(* CODESYS project DCCM PLC 1.project
   Author: jrfsc
   Version: 0.0.0.0
   Title: DCCM PLC 1

Project tree, tasks and I/O mapping:
  DCCM_PLC_1 : TM251MESC, Schneider Electric, order no. TM251MESC, version 5.1.9.35
      settings: OPCUA enable = False
    application Application
      libraries: SysTimeRtc, * (System); CAA Memory, 3.5.12.0 (CAA Technical Workgroup); IecRtsServices, 1.0.4.0 (Schneider Electric)
      task MAST (cyclic, interval 20 ms, priority 15, watchdog 100 ms x 1) calls INPUT_MAPPING, FILTER_ALARMS, FAN_2STAGES_FAULT_DETECTION, DEPROX_COUNT, FAN_2STAGES, PandemicCheck, DAMPER_CONTROL, SR_Main, OUTPUT_MAPPING
      global variables GVL
      program SR_Main [FBD]
      program INPUT_MAPPING [ST]
      program OUTPUT_MAPPING [ST]
      FBs/
        function block DUTY [ST]
        function block DUTY_CHANGE [ST]
        function block FB_9StatesMonitoring [ST]
        function block FB_DUTY_DUTY_STANDBY_PUMP_SPD [ST]
        function block FB_FLOATING_VALVE [ST]
        function block FB_HEATING_OR_COOLING [ST]
        function block FB_OMODE [ST]
        function block FB_PMODE [ST]
        function block FB_SETPOINT_MODE [ST]
        function block FB_WATCHDOG [ST]
        function block LINEAR [ST]
        function block SATSP_CALC [ST]
        function block SB_HEATING_COOLING [ST]
        function block TERMINAL_LOAD [ST]
        function block FB_0_10V_TO_2_10V_OUTPUT [ST]
        function block FB_2STAGES_DUTY [ST]
        function block FB_DUTYTRIGGER [ST]
        function block FB_FanProvingSwitchOverEnable [ST]
        function block FB_2STAGES_DUTY_1 [ST]
        function block SWITCH_CHECK [ST]
      Enumeration/
        data type ET_9STATE_MONITORING
        data type ET_OMODE
        data type ET_PMODE
      LIBRARY/
        function block FB_PULSE_GENERATOR [ST]
      Library/
        function block FB_SETPOINT_RAMPING [ST]
        function block FB_PCMS_WATCHDOG [ST]
      program SYSTEM_DATE_TIME [ST]
      program DAMPER_CONTROL [FBD]
      program FILTER_ALARMS [FBD]
      program DEPROX_COUNT [CFC]
      program FAN_2STAGES [FBD]: ACT_GetCurrentDateTime
      program FAN_2STAGES_FAULT_DETECTION [FBD]
      global variables PersistentVars
      program PandemicCheck [CFC]
    IO_Bus : IO bus - TM3, Schneider Electric, version 5.1.9.35
      Module_1 : TM3AQ4/G, Schneider Electric, order no. TM3AQ4/G, version 1.0.0.16
          settings: KPI Configuration.KPI Configuration = 16; KPI Configuration.KPI Configuration = 0; KPI Configuration.KPI Configuration = 16; KPI Configuration.KPI Configuration = 39
          output qPLANT_EXHAUST_DAMPER : INT  // QW0
          output qiModule_1_QW3 : INT  // QW3
          input  ibModule_1_IBStatusQW0 : BYTE  // IBStatusQW0
          input  ibModule_1_IBStatusQW1 : BYTE  // IBStatusQW1
          input  ibModule_1_IBStatusQW2 : BYTE  // IBStatusQW2
          input  ibModule_1_IBStatusQW3 : BYTE  // IBStatusQW3
          unmapped channels: QW1, QW2
      Module_2 : TM3AI8/G, Schneider Electric, order no. TM3AI8/G, version 1.0.0.27
          settings: KPI Configuration.KPI Configuration = 32; KPI Configuration.KPI Configuration = 32; KPI Configuration.KPI Configuration = 32; KPI Configuration.KPI Configuration = 32; KPI Configuration.KPI Configuration = 32; KPI Configuration.KPI Configuration = 32; KPI Configuration.KPI Configuration = 32; KPI Configuration.KPI Configuration = 32; KPI Configuration.KPI Configuration = 0; KPI Configuration.KPI Configuration = 0; KPI Configuration.KPI Configuration = 0; KPI Configuration.KPI Configuration = 0; KPI Configuration.KPI Configuration = 0; KPI Configuration.KPI Configuration = 0; KPI Configuration.KPI Configuration = 0; KPI Configuration.KPI Configuration = 0; KPI Configuration.KPI Configuration = 50; KPI Configuration.KPI Configuration = 0; KPI Configuration.KPI Configuration = 250; KPI Configuration.KPI Configuration = 0; KPI Configuration.KPI Configuration = 250; KPI Configuration.KPI Configuration = 0; KPI Configuration.KPI Configuration = 250; KPI Configuration.KPI Configuration = 0; KPI Configuration.KPI Configuration = 244; KPI Configuration.KPI Configuration = 1; KPI Configuration.KPI Configuration = 244; KPI Configuration.KPI Configuration = 1; KPI Configuration.KPI Configuration = 244; KPI Configuration.KPI Configuration = 1; KPI Configuration.KPI Configuration = 16; KPI Configuration.KPI Configuration = 39; KPI Configuration.KPI Configuration = 100
          input  iEXHAUST_AIR_VELOCITY : INT  // IW0
          input  iPREFILTER1_DP : INT  // IW1
          input  iPREFILTER2_DP : INT  // IW2
          input  iPREFILTER3_DP : INT  // IW3
          input  iHEPA1_DP : INT  // IW4
          input  iHEPA2_DP : INT  // IW5
          input  iHEPA3_DP : INT  // IW6
          input  iPLANT_EXHAUST_DAMPER_STS : INT  // IW7
          input  ibModule_2_IBStatusIW0 : BYTE  // IBStatusIW0
          input  ibModule_2_IBStatusIW1 : BYTE  // IBStatusIW1
          input  ibModule_2_IBStatusIW2 : BYTE  // IBStatusIW2
          input  ibModule_2_IBStatusIW3 : BYTE  // IBStatusIW3
          input  ibModule_2_IBStatusIW4 : BYTE  // IBStatusIW4
          input  ibModule_2_IBStatusIW5 : BYTE  // IBStatusIW5
          input  ibModule_2_IBStatusIW6 : BYTE  // IBStatusIW6
          input  ibModule_2_IBStatusIW7 : BYTE  // IBStatusIW7
      Module_3 : TM3DM24R/G, Schneider Electric, order no. TM3DM24R/G, version 1.0.2.0
          input  iPRESSURE_SWITCH1 : BOOL  // IW0.I0
          input  iPRESSURE_SWITCH2 : BOOL  // IW0.I1
          input  iFAN1_MANUAL_SW : BOOL  // IW0.I2
          input  iFAN1_AUTO_SW : BOOL  // IW0.I3
          input  iFAN2_MANUAL_SW : BOOL  // IW0.I4
          input  iFAN2_AUTO_SW : BOOL  // IW0.I5
          input  iFAN1_READY : BOOL  // IW0.I6
          input  iFAN1_RUN : BOOL  // IW0.I7
          input  iFAN1_FAULT : BOOL  // IW0.I8
          input  iFAN2_READY : BOOL  // IW0.I9
          input  iFAN2_RUN : BOOL  // IW0.I10
          input  iFAN2_FAULT : BOOL  // IW0.I11
          input  iFIRE_DAMPER_STS : BOOL  // IW0.I12
          input  iDISCHARGE_DAMPER1_STS : BOOL  // IW0.I13
          input  iDISCHARGE_DAMPER2_STS : BOOL  // IW0.I14
          input  iRETURN_DAMPER1_STS : BOOL  // IW0.I15
          output qFAN1_SS : BOOL  // QB0.Q0
          output qFAN2_SS : BOOL  // QB0.Q1
          output qFAN1_DISCHARGE_DAMPER : BOOL  // QB0.Q2
          output qFAN2_DISCHARGE_DAMPER : BOOL  // QB0.Q3
          output qPLANT_RETURN_DAMPER : BOOL  // QB0.Q4
          unmapped channels: IW0, QB0
      Module_4 : TM3AM6/G, Schneider Electric, order no. TM3AM6/G, version 1.0.0.23
          settings: KPI Configuration.KPI Configuration = 32; KPI Configuration.KPI Configuration = 32; KPI Configuration.KPI Configuration = 0; KPI Configuration.KPI Configuration = 0; KPI Configuration.KPI Configuration = 16; KPI Configuration.KPI Configuration = 39; KPI Configuration.KPI Configuration = 16; KPI Configuration.KPI Configuration = 39; KPI Configuration.KPI Configuration = 16; KPI Configuration.KPI Configuration = 16; KPI Configuration.KPI Configuration = 0; KPI Configuration.KPI Configuration = 0; KPI Configuration.KPI Configuration = 16; KPI Configuration.KPI Configuration = 39; KPI Configuration.KPI Configuration = 16; KPI Configuration.KPI Configuration = 39
          input  iFAN1_SPDFB : INT  // IW0
          input  iFAN2_SPDFB : INT  // IW1
          input  iiModule_4_IW2 : INT  // IW2
          input  iiModule_4_IW3 : INT  // IW3
          output qFAN1_SPD : INT  // QW0
          output qFAN2_SPD : INT  // QW1
          input  ibModule_4_IBStatusIW0 : BYTE  // IBStatusIW0
          input  ibModule_4_IBStatusIW1 : BYTE  // IBStatusIW1
          input  ibModule_4_IBStatusIW2 : BYTE  // IBStatusIW2
          input  ibModule_4_IBStatusIW3 : BYTE  // IBStatusIW3
          input  ibModule_4_IBStatusQW0 : BYTE  // IBStatusQW0
          input  ibModule_4_IBStatusQW1 : BYTE  // IBStatusQW1
    COM_Bus : COM bus, Schneider Electric, version 5.1.9.35
    Ethernet_1 : Ethernet Network, Schneider Electric, version 5.1.9.35
        settings: WebServer = TRUE; FTP Server = FALSE; SoMachine Protocol = TRUE; Modbus Server = TRUE; NetManage Protocol = TRUE; SNMP protocol = FALSE; WebVisu protocol = FALSE; Secured Web Server = TRUE
    Serial_Line_1 : Serial line, Schneider Electric, version 5.1.9.35
      Machine_Expert_Network_Manager : Machine Expert-Network Manager, Schneider Electric, version 4.0.0.4
    CAN_1 : CANopen bus, Schneider Electric, version 5.1.9.35
  FdtConnections : FDT Connections, Schneider Electric, version 1.0.0.2
*)

// DCCM_PLC_1/Application/Enumeration/ET_9STATE_MONITORING
{attribute 'qualified_only' := ''}
{attribute 'strict' := ''}
TYPE ET_9STATE_MONITORING :
(
	STOPPED := 0,
	RUNNING := 1,
	STARTING := 2,
	STOPPING := 3,
	START_FAIL := 4,
	STOP_FAIL := 5,
	UNEXPECTED_START := 6,
	UNEXPECTED_STOP := 7,
	FIRE_STOP := 8,
	UNKNOWN := 9
);
END_TYPE

// DCCM_PLC_1/Application/Enumeration/ET_OMODE
{attribute 'qualified_only' := ''}
{attribute 'strict' := ''}
TYPE ET_OMODE :
(
	UNOCC := 0,
	OPTSTART := 1,
	SCH := 2,
	AHRS := 3,
	MOTDETECT := 4,
	SETBACK := 7
);
END_TYPE

// DCCM_PLC_1/Application/Enumeration/ET_PMODE
{attribute 'qualified_only' := ''}
{attribute 'strict' := ''}
TYPE ET_PMODE :
(
	OFF_NORMAL := 0,
	OFF_PCMS := 1,
	OFF_Fire := 2,
	OFF_DMPRLOCK := 3,
	OFF_RESET := 4,
	Startup := 5,
	Purge := 6,
	RUN_NORMAL := 7
);
END_TYPE

// DCCM_PLC_1/Application/GVL
{attribute 'qualified_only'}
VAR_GLOBAL
	FAN1_SPEED AT %MD500: REAL;
	FAN2_SPEED AT %MD501: REAL;
	COMMS_ERROR_ROOM AT %MX6.1: BOOL;
	FAN2_FB AT %MD534: REAL;
	FAN1_FB AT %MD533: REAL;
	FAN1_SWITCH_TOTAL AT %MW9006: INT;
	FAN2_SWITCH_TOTAL AT %MW9007: INT;
	fan2SS_del: BOOL;
	fan1SS_del: bool;
	VEL_PRESS_LITRES AT %MD536: REAL;
	FAN2_FAULT_RESET AT %MX5.7: BOOL;
	FAN1_FAULT_RESET AT %MX5.6: BOOL;
END_VAR
VAR_GLOBAL RETAIN PERSISTENT
	EXHAUST_VEL_PRESS_SP AT %MD502: REAL := 3;
END_VAR
VAR_GLOBAL
	PREFILTER1_DP AT %MD503: REAL;
	PREFILTER2_DP AT %MD504: REAL;
	PREFILTER3_DP AT %MD505: REAL;
	HEPA1_DP AT %MD506: REAL;
	HEPA2_DP AT %MD507: REAL;
	HEPA3_DP AT %MD508: REAL;
	PRESSURE_SWITCH1 AT %MX0.0: BOOL;
	PRESSURE_SWITCH2 AT %MX0.1: BOOL;
	FAN1_MANUAL_SW AT %MX0.2: BOOL;
	FAN1_AUTO_SW AT %MX0.3: BOOL;
	FAN2_MANUAL_SW AT %MX0.4: BOOL;
	FAN2_AUTO_SW AT %MX0.5: BOOL;
	FAN1_READY AT %MX0.6: BOOL;
	FAN1_RUN AT %MX0.7: BOOL;
	FAN1_FAULT AT %MX1.0: BOOL;
	FAN2_READY AT %MX1.1: BOOL;
	FAN2_RUN AT %MX1.2: BOOL;
	FAN2_FAULT AT %MX1.3: BOOL;
	FIRE AT %MX1.4: BOOL;
	DISCHARGE_DAMPER1_STS AT %MX1.5: BOOL;
	DISCHARGE_DAMPER2_STS AT %MX1.6: BOOL;
	FAN1_SS AT %MX1.7: BOOL;
	FAN2_SS AT %MX2.0: BOOL;
	FAN1_DISCHARGE_DAMPER AT %MX2.1: BOOL;
	FAN2_DISCHARGE_DAMPER AT %MX2.2: BOOL;
	SYS_HOUR: UINT;
	SYS_DAY: UINT;
	SYS_MINUTE: UINT;
END_VAR
VAR_GLOBAL RETAIN PERSISTENT
	STANDBY_FAN_NO AT %MW9002: INT := 2;
	STANDBY_FAN_NO_MANUAL AT %MW9003: INT := 1;
	STANDBY_FAN_NO_MODE AT %MX2.5: BOOL := 1;
	FAN1_SS_MANUAL AT %MX2.6: BOOL;
	FAN1_SS_MODE AT %MX2.7: BOOL;
	FAN2_SS_MANUAL AT %MX3.0: BOOL;
	FAN2_SS_MODE AT %MX3.1: BOOL;
END_VAR
VAR_GLOBAL
	EXHAUST_VEL_PRESS AT %MD509: REAL;
END_VAR
VAR_GLOBAL RETAIN PERSISTENT
	FAN1_SPEED_MANUAL AT %MD510: REAL;
	FAN1_SPEED_MODE AT %MX3.2: BOOL;
	FAN2_SPEED_MANUAL AT %MD511: REAL;
	FAN2_SPEED_MODE AT %MX4.5: BOOL;
END_VAR
VAR_GLOBAL
	ISO_MD1 AT %MD527: REAL;
END_VAR
VAR_GLOBAL RETAIN PERSISTENT
	EF_VEL_PRESS_SP1 AT %MD512: REAL := 2;
	FAN1_DISCHARGE_DAMPER_MAN AT %MX3.3: BOOL;
	FAN1_DISCHARGE_DAMPER_MD AT %MX3.4: BOOL;
	FAN2_DISCHARGE_DAMPER_MAN AT %MX3.5: BOOL;
	FAN2_DISCHARGE_DAMPER_MD AT %MX3.6: BOOL;
END_VAR
VAR_GLOBAL
	FAN1_ST_MONITORING AT %MW9001: UINT;
	FAN2_ST_MONITORING AT %MW9004: UINT;
END_VAR
VAR_GLOBAL RETAIN PERSISTENT
	PREFILTER1_ALMSP AT %MD513: REAL;
	PREFILTER2_ALMSP AT %MD514: REAL;
	PREFILTER3_ALMSP AT %MD515: REAL;
	HEPA1_ALMSP AT %MD516: REAL;
	HEPA2_ALMSP AT %MD517: REAL;
	HEPA3_ALMSP AT %MD518: REAL;
END_VAR
VAR_GLOBAL
	PREFILTER1_ALM AT %MX3.7: BOOL;
	PREFILTER2_ALM AT %MX4.0: BOOL;
	PREFILTER3_ALM AT %MX4.1: BOOL;
	HEPA1_ALM AT %MX4.2: BOOL;
	HEPA2_ALM AT %MX4.3: BOOL;
	HEPA3_ALM AT %MX4.4: BOOL;
	ISO_MD2 AT %MD524: REAL;
	ISO_MD3 AT %MD525: REAL;
	ISO_MD4 AT %MD526: REAL;
	ISO_MD1_DW: REAL;
	ISO_MD2_DW: REAL;
	ISO_MD3_DW: REAL;
	ISO_MD4_DW: REAL;
END_VAR
VAR_GLOBAL RETAIN PERSISTENT
	PLANT_EXHAUST_DAMPER AT %MD523: REAL;
	PLANT_RETURN_DAMPER AT %MX5.2: BOOL;
	PLANT_RETURN_DAMPER_STS AT %MX5.1: BOOL;
END_VAR
VAR_GLOBAL
	PLANT_EXHAUST_DAMPER_STS AT %MD522: REAL;
END_VAR
VAR_GLOBAL RETAIN PERSISTENT
	PLANT_RETURN_DAMPER_MAN AT %MX5.0: BOOL;
	PLANT_RETURN_DAMPER_MD AT %MX5.5: BOOL;
	PLANT_RETURN_DAMPER_SS AT %MX5.4: BOOL;
	PLANT_EXHAUST_DAMPER_MD AT %MX5.3: BOOL;
	PLANT_EXHAUST_DAMPER_MAN AT %MD520: REAL;
	PLANT_EXHAUST_DAMPER_PAN AT %MD535: REAL;
	PLANT_EXHAUST_DAMPER_SP AT %MD521: REAL := 100;
	EF_VEL_PRESS_SP2 AT %MD528: REAL := 2;
	EF_VEL_PRESS_SP3 AT %MD529: REAL := 2;
	EF_VEL_PRESS_SP4 AT %MD530: REAL := 0;
	FAN_PID_P AT %MD532: REAL;
	FAN_PID_I AT %MD531: REAL;
	EXHAUST_VEL_PRESS_PAN_SP AT %MD550: REAL := 16;
	EXHAUST_VEL_PRESS_PAN_SP1 AT %MD551: REAL := 14;
	EXHAUST_VEL_PRESS_PAN_SP2 AT %MD552: REAL := 10;
	EXHAUST_VEL_PRESS_PAN_SP3 AT %MD553: REAL := 8;
	EXHAUST_VEL_PRESS_PAN_SP4 AT %MD554: REAL := 0;
END_VAR
VAR_GLOBAL
	OPEN_DAMPER1: BOOL;
	OPEN_DAMPER2: BOOL;
	FAN1_ST: BOOL;
	FAN2_ST: BOOL;
	PANDEMIC AT %MW9005: INT;
	COMMS_ERROR: BOOL;
	newVarGlobal: BOOL;
	COMMS_ERROR_AHU AT %MX6.0: BOOL;
END_VAR

// DCCM_PLC_1/Application/PersistentVars
{attribute 'qualified_only'}
VAR_GLOBAL PERSISTENT RETAIN
	// Generated instance path of persistent variable
	GVL.EXHAUST_VEL_PRESS_SP: REAL;
	// Generated instance path of persistent variable
	GVL.STANDBY_FAN_NO: INT := INT#2;
	// Generated instance path of persistent variable
	GVL.STANDBY_FAN_NO_MANUAL: INT := INT#1;
	// Generated instance path of persistent variable
	GVL.STANDBY_FAN_NO_MODE: BOOL := TRUE;
	// Generated instance path of persistent variable
	GVL.FAN1_SS_MANUAL: BOOL;
	// Generated instance path of persistent variable
	GVL.FAN1_SS_MODE: BOOL;
	// Generated instance path of persistent variable
	GVL.FAN2_SS_MANUAL: BOOL;
	// Generated instance path of persistent variable
	GVL.FAN2_SS_MODE: BOOL;
	// Generated instance path of persistent variable
	GVL.FAN1_SPEED_MANUAL: REAL;
	// Generated instance path of persistent variable
	GVL.FAN1_SPEED_MODE: BOOL;
	// Generated instance path of persistent variable
	GVL.FAN2_SPEED_MANUAL: REAL;
	// Generated instance path of persistent variable
	GVL.FAN2_SPEED_MODE: BOOL;
	// Generated instance path of persistent variable
	GVL.EF_VEL_PRESS_SP1: REAL;
	// Generated instance path of persistent variable
	GVL.FAN1_DISCHARGE_DAMPER_MAN: BOOL;
	// Generated instance path of persistent variable
	GVL.FAN1_DISCHARGE_DAMPER_MD: BOOL;
	// Generated instance path of persistent variable
	GVL.FAN2_DISCHARGE_DAMPER_MAN: BOOL;
	// Generated instance path of persistent variable
	GVL.FAN2_DISCHARGE_DAMPER_MD: BOOL;
	// Generated instance path of persistent variable
	GVL.PREFILTER1_ALMSP: REAL;
	// Generated instance path of persistent variable
	GVL.PREFILTER2_ALMSP: REAL;
	// Generated instance path of persistent variable
	GVL.PREFILTER3_ALMSP: REAL;
	// Generated instance path of persistent variable
	GVL.HEPA1_ALMSP: REAL;
	// Generated instance path of persistent variable
	GVL.HEPA2_ALMSP: REAL;
	// Generated instance path of persistent variable
	GVL.HEPA3_ALMSP: REAL;
	// Generated instance path of persistent variable
	GVL.PLANT_EXHAUST_DAMPER: REAL;
	// Generated instance path of persistent variable
	GVL.PLANT_RETURN_DAMPER: BOOL;
	// Generated instance path of persistent variable
	GVL.PLANT_RETURN_DAMPER_STS: BOOL;
	// Generated instance path of persistent variable
	GVL.PLANT_RETURN_DAMPER_MAN: BOOL;
	// Generated instance path of persistent variable
	GVL.PLANT_RETURN_DAMPER_MD: BOOL;
	// Generated instance path of persistent variable
	GVL.PLANT_RETURN_DAMPER_SS: BOOL;
	// Generated instance path of persistent variable
	GVL.PLANT_EXHAUST_DAMPER_MD: BOOL;
	// Generated instance path of persistent variable
	GVL.PLANT_EXHAUST_DAMPER_MAN: REAL;
	// Generated instance path of persistent variable
	GVL.PLANT_EXHAUST_DAMPER_PAN: REAL;
	// Generated instance path of persistent variable
	GVL.PLANT_EXHAUST_DAMPER_SP: REAL := 100.0;
	// Generated instance path of persistent variable
	GVL.EF_VEL_PRESS_SP2: REAL;
	// Generated instance path of persistent variable
	GVL.EF_VEL_PRESS_SP3: REAL;
	// Generated instance path of persistent variable
	GVL.EF_VEL_PRESS_SP4: REAL;
	// Generated instance path of persistent variable
	GVL.FAN_PID_P: REAL;
	// Generated instance path of persistent variable
	GVL.FAN_PID_I: REAL;
END_VAR

// DCCM_PLC_1/Application/INPUT_MAPPING
PROGRAM INPUT_MAPPING
VAR

	voltage_converter: FB_0_10V_TO_2_10V_OUTPUT;
END_VAR

//MAPPINGHARDWARE INPUTS TO MEMORY WORDS

GVL.EXHAUST_VEL_PRESS := TO_REAL(iEXHAUST_AIR_VELOCITY);								//MODULE 2 TM3AI8 INPUT 0

GVL.VEL_PRESS_LITRES := GVL.EXHAUST_VEL_PRESS*81.9;

GVL.PREFILTER1_DP := TO_REAL(iPREFILTER1_DP);											//MODULE 2 TM3AI8 INPUT 1
GVL.PREFILTER2_DP := TO_REAL(iPREFILTER2_DP);											//MODULE 2 TM3AI8 INPUT 2
GVL.PREFILTER3_DP := TO_REAL(iPREFILTER3_DP);											//MODULE 2 TM3AI8 INPUT 3
GVL.HEPA1_DP := TO_REAL(iHEPA1_DP);														//MODULE 2 TM3AI8 INPUT 4
GVL.HEPA2_DP := TO_REAL(iHEPA2_DP);														//MODULE 2 TM3AI8 INPUT 5
GVL.HEPA3_DP := TO_REAL(iHEPA3_DP);														//MODULE 2 TM3AI8 INPUT 6

GVL.PRESSURE_SWITCH1 := iPRESSURE_SWITCH1;												//MODULE 3 TM3DM24R INPUT 0
GVL.PRESSURE_SWITCH2 := iPRESSURE_SWITCH2;												//MODULE 3 TM3DM24R INPUT 1

GVL.FAN1_MANUAL_SW := iFAN1_MANUAL_SW;													//MODULE 3 TM3DM24R INPUT 2
GVL.FAN1_AUTO_SW := iFAN1_AUTO_SW;														//MODULE 3 TM3DM24R INPUT 3

GVL.FAN2_MANUAL_SW := iFAN2_MANUAL_SW;													//MODULE 3 TM3DM24R INPUT 4
GVL.FAN2_AUTO_SW := iFAN2_AUTO_SW;														//MODULE 3 TM3DM24R INPUT 5


GVL.FAN1_READY := iFAN1_READY;															//MODULE 3 TM3DM24R INPUT 6
GVL.FAN1_RUN := iFAN1_RUN;																//MODULE 3 TM3DM24R INPUT 7
GVL.FAN1_FAULT := iFAN1_FAULT;															//MODULE 3 TM3DM24R INPUT 8
GVL.FAN2_READY := iFAN2_READY;															//MODULE 3 TM3DM24R INPUT 9
GVL.FAN2_RUN := iFAN2_RUN;																//MODULE 3 TM3DM24R INPUT 10
GVL.FAN2_FAULT := iFAN2_FAULT;															//MODULE 3 TM3DM24R INPUT 11

GVL.FIRE := iFIRE_DAMPER_STS;													//MODULE 3 TM3DM24R INPUT 12
GVL.DISCHARGE_DAMPER1_STS := iDISCHARGE_DAMPER1_STS;									//MODULE 3 TM3DM24R INPUT 13
GVL.DISCHARGE_DAMPER2_STS := iDISCHARGE_DAMPER2_STS;									//MODULE 3 TM3DM24R INPUT 14


GVL.PLANT_EXHAUST_DAMPER_STS:=100-(((((iPLANT_EXHAUST_DAMPER_STS/100)-100) * 100/80))+100);

GVL.OPEN_DAMPER1 := (GVL.FAN1_ST_MONITORING = ET_9STATE_MONITORING.RUNNING)OR(GVL.FAN1_ST_MONITORING = ET_9STATE_MONITORING.STOP_FAIL)OR(GVL.FAN1_ST_MONITORING = ET_9STATE_MONITORING.UNEXPECTED_START)OR(GVL.FAN1_ST_MONITORING = ET_9STATE_MONITORING.STARTING);
GVL.OPEN_DAMPER2 := (GVL.FAN2_ST_MONITORING = ET_9STATE_MONITORING.RUNNING)OR(GVL.FAN2_ST_MONITORING = ET_9STATE_MONITORING.STOP_FAIL)OR(GVL.FAN2_ST_MONITORING = ET_9STATE_MONITORING.UNEXPECTED_START)OR(GVL.FAN2_ST_MONITORING = ET_9STATE_MONITORING.STARTING);
				
GVL.PLANT_RETURN_DAMPER_STS := NOT(iRETURN_DAMPER1_STS);	 //True=OPEN			

GVL.FAN1_ST := (iFAN1_SPDFB > 200);  //AI2
GVL.FAN2_ST := (iFAN2_SPDFB > 200); //AI3

GVL.FAN1_FB := iFAN1_SPDFB/100;  //AI2
GVL.FAN2_FB := iFAN2_SPDFB/100; //AI3

END_PROGRAM

// DCCM_PLC_1/Application/FBs/FB_0_10V_TO_2_10V_OUTPUT
FUNCTION_BLOCK FB_0_10V_TO_2_10V_OUTPUT
VAR_OUTPUT
	// 0-10V = 0-100%
	OUT_PRCT: REAL;
END_VAR
VAR_INPUT
	// 2-10V = 0-100%
	IN_PRCT: REAL;
END_VAR

OUT_PRCT := ((IN_PRCT * 0.08) + 2) * 10;

END_FUNCTION_BLOCK

// DCCM_PLC_1/Application/FILTER_ALARMS
PROGRAM FILTER_ALARMS
VAR
	TON_0: TON;
	TON_1: TON;
	TON_2: TON;
	TON_3: TON;
	TON_4: TON;
	TON_5: TON;
END_VAR

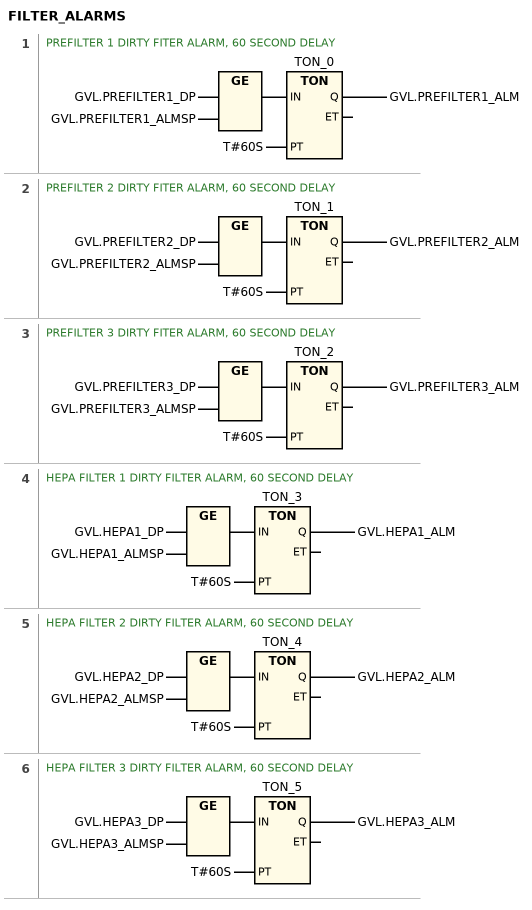
// NETWORK 1
// PREFILTER 1 DIRTY FITER ALARM, 60 SECOND DELAY
TON_0(IN := GVL.PREFILTER1_DP >= GVL.PREFILTER1_ALMSP, PT := T#60S); // TON
GVL.PREFILTER1_ALM := TON_0.Q;

// NETWORK 2
// PREFILTER 2 DIRTY FITER ALARM, 60 SECOND DELAY
TON_1(IN := GVL.PREFILTER2_DP >= GVL.PREFILTER2_ALMSP, PT := T#60S); // TON
GVL.PREFILTER2_ALM := TON_1.Q;

// NETWORK 3
// PREFILTER 3 DIRTY FITER ALARM, 60 SECOND DELAY
TON_2(IN := GVL.PREFILTER3_DP >= GVL.PREFILTER3_ALMSP, PT := T#60S); // TON
GVL.PREFILTER3_ALM := TON_2.Q;

// NETWORK 4
// HEPA FILTER 1 DIRTY FILTER ALARM, 60 SECOND DELAY
TON_3(IN := GVL.HEPA1_DP >= GVL.HEPA1_ALMSP, PT := T#60S); // TON
GVL.HEPA1_ALM := TON_3.Q;

// NETWORK 5
// HEPA FILTER 2 DIRTY FILTER ALARM, 60 SECOND DELAY
TON_4(IN := GVL.HEPA2_DP >= GVL.HEPA2_ALMSP, PT := T#60S); // TON
GVL.HEPA2_ALM := TON_4.Q;

// NETWORK 6
// HEPA FILTER 3 DIRTY FILTER ALARM, 60 SECOND DELAY
TON_5(IN := GVL.HEPA3_DP >= GVL.HEPA3_ALMSP, PT := T#60S); // TON
GVL.HEPA3_ALM := TON_5.Q;

END_PROGRAM

// DCCM_PLC_1/Application/FAN_2STAGES_FAULT_DETECTION
PROGRAM FAN_2STAGES_FAULT_DETECTION
VAR
	FAN1_MONITOR: FB_9StatesMonitoring;
	FAN2_MONITOR: FB_9StatesMonitoring;
	TOF_0: TOF;
	TON_0: TON;
	TON_1: TON;
	tom_2: TON;
	TON_2: TON;
	TON_3: TON;
	FAN2_FAULT_LATCH: RS;
	FAN1_FAULT_LATCH: RS;
END_VAR

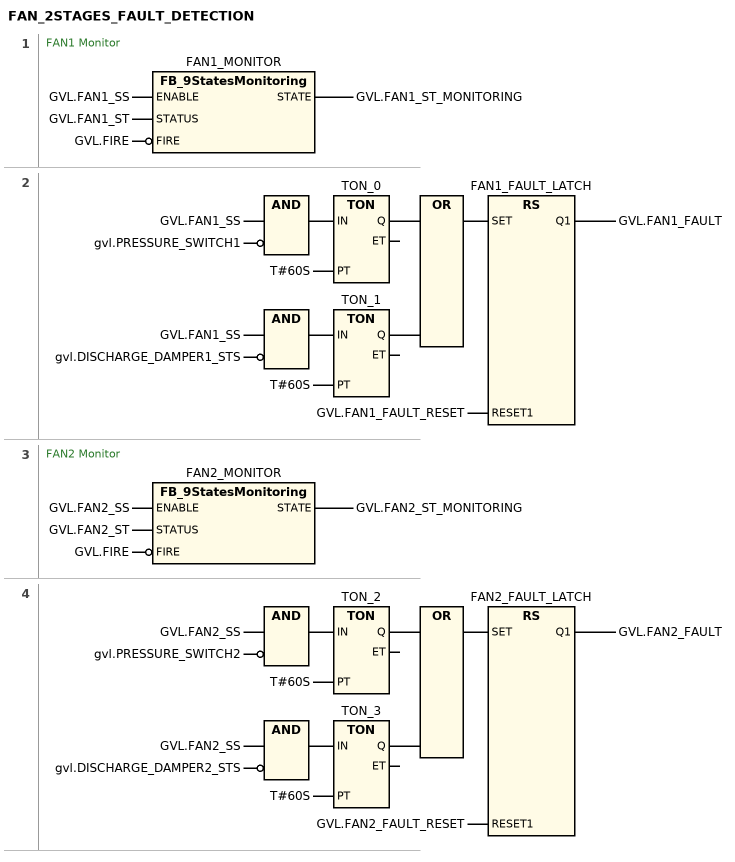
// NETWORK 1
// FAN1 Monitor
FAN1_MONITOR(ENABLE := GVL.FAN1_SS, STATUS := GVL.FAN1_ST, FIRE := NOT GVL.FIRE); // FB_9StatesMonitoring
GVL.FAN1_ST_MONITORING := FAN1_MONITOR.STATE;

// NETWORK 2
TON_0(IN := GVL.FAN1_SS AND NOT gvl.PRESSURE_SWITCH1, PT := T#60S); // TON
TON_1(IN := GVL.FAN1_SS AND NOT gvl.DISCHARGE_DAMPER1_STS, PT := T#60S); // TON
FAN1_FAULT_LATCH(SET := TON_0.Q OR TON_1.Q, RESET1 := GVL.FAN1_FAULT_RESET); // RS
GVL.FAN1_FAULT := FAN1_FAULT_LATCH.Q1;

// NETWORK 3
// FAN2 Monitor
FAN2_MONITOR(ENABLE := GVL.FAN2_SS, STATUS := GVL.FAN2_ST, FIRE := NOT GVL.FIRE); // FB_9StatesMonitoring
GVL.FAN2_ST_MONITORING := FAN2_MONITOR.STATE;

// NETWORK 4
TON_2(IN := GVL.FAN2_SS AND NOT gvl.PRESSURE_SWITCH2, PT := T#60S); // TON
TON_3(IN := GVL.FAN2_SS AND NOT gvl.DISCHARGE_DAMPER2_STS, PT := T#60S); // TON
FAN2_FAULT_LATCH(SET := TON_2.Q OR TON_3.Q, RESET1 := GVL.FAN2_FAULT_RESET); // RS
GVL.FAN2_FAULT := FAN2_FAULT_LATCH.Q1;

END_PROGRAM

// DCCM_PLC_1/Application/FBs/FB_9StatesMonitoring
FUNCTION_BLOCK FB_9StatesMonitoring
VAR
	ENABLE_OFF: BOOL := FALSE;
	ENABLE_ON: BOOL := FALSE;
	STATUS_ON: BOOL := FALSE;
	STATUS_OFF: BOOL := FALSE;
	FIRE_ON: BOOL := FALSE;
	FIRE_OFF: BOOL := FALSE;
	BEEN_RUNNING_OK: BOOL := FALSE;
	NOT_BEEN_RUNNING_OK: BOOL := FALSE;
	ALL_OFF: BOOL := FALSE;
	NOT_ALL_OFF: BOOL := FALSE;
	START_DELAY_ON: BOOL := FALSE;
	START_DELAY_OFF: BOOL := FALSE;
	STOP_DELAY_ON: BOOL := FALSE;
	STOP_DELAY_OFF: BOOL := FALSE;
	ENABLE_TIMER_ON: BOOL := FALSE;
	ENABLE_TIMER_OFF: BOOL := FALSE;
	BEEN_RUNNING_OK_LATCH: RS;
	ALL_OFF_LATCH: RS;
	START_DELAY_TON: TON;
	STOP_DELAY_TON: TON;
	STOPPED: INT;
END_VAR
VAR_INPUT
	ENABLE: BOOL := FALSE;
	STATUS: BOOL := FALSE;
	FIRE: BOOL := FALSE;
END_VAR
VAR_OUTPUT
	STATE: ET_9STATE_MONITORING := 9;
END_VAR

(* 
Version 1.0
Last Updated: 28/01/2020

9 States Monitoring. Value from 0 to 9
	STOPPED := 0,
	RUNNING := 1,
	STARTING := 2,
	STOPPING := 3,
	START_FAIL := 4,
	STOP_FAIL := 5,
	UNEXPECTED_START := 6,
	UNEXPECTED_STOP := 7,
	FIRE_STOP := 8,
	UNKNOWN := 9
*)

ENABLE_OFF := (ENABLE = FALSE);
ENABLE_ON := (ENABLE = TRUE);
STATUS_ON := (STATUS = TRUE);
STATUS_OFF := (STATUS = FALSE);
FIRE_ON := (FIRE = TRUE);
FIRE_OFF := (FIRE = FALSE);

BEEN_RUNNING_OK_LATCH(SET := ENABLE_ON AND STATUS_ON, RESET1 := ENABLE_OFF);
BEEN_RUNNING_OK := BEEN_RUNNING_OK_LATCH.Q1;

ALL_OFF_LATCH(SET := ENABLE_OFF AND STATUS_OFF, RESET1 := ENABLE_ON);
ALL_OFF := ALL_OFF_LATCH.Q1;

START_DELAY_TON(IN := ENABLE_ON, PT := T#30S);
START_DELAY_ON := START_DELAY_TON.Q;

STOP_DELAY_TON(IN := ENABLE_OFF, PT := T#30S);
STOP_DELAY_ON := STOP_DELAY_TON.Q;

ENABLE_TIMER_ON := ((START_DELAY_TON.ET < T#30S AND ENABLE_ON) OR (STOP_DELAY_TON.ET < T#30S AND ENABLE_OFF));

START_DELAY_OFF := NOT START_DELAY_ON;
STOP_DELAY_OFF := NOT STOP_DELAY_ON;
ENABLE_TIMER_OFF := NOT ENABLE_TIMER_ON;
NOT_BEEN_RUNNING_OK := NOT BEEN_RUNNING_OK;
NOT_ALL_OFF := NOT ALL_OFF;

IF (ENABLE_ON AND STATUS_OFF AND FIRE_ON) THEN
	STATE := ET_9STATE_MONITORING.FIRE_STOP;
ELSIF (ENABLE_OFF AND STATUS_ON AND STOP_DELAY_ON AND NOT_BEEN_RUNNING_OK AND NOT_ALL_OFF) THEN
	STATE := ET_9STATE_MONITORING.STOP_FAIL;
ELSIF (ENABLE_ON AND STATUS_OFF AND START_DELAY_ON AND NOT_BEEN_RUNNING_OK AND NOT_ALL_OFF) THEN
	STATE := ET_9STATE_MONITORING.START_FAIL;
ELSIF (ENABLE_OFF AND STATUS_ON AND ENABLE_TIMER_OFF AND STOP_DELAY_ON AND ENABLE_TIMER_OFF AND ALL_OFF) THEN
	STATE := ET_9STATE_MONITORING.UNEXPECTED_START;
ELSIF (ENABLE_ON AND STATUS_OFF AND START_DELAY_ON AND FIRE_OFF AND ENABLE_TIMER_OFF AND BEEN_RUNNING_OK AND NOT_ALL_OFF) THEN
	STATE := ET_9STATE_MONITORING.UNEXPECTED_STOP;
ELSIF (ENABLE_OFF AND STATUS_ON AND ENABLE_TIMER_ON AND STOP_DELAY_OFF AND FIRE_OFF) THEN
	STATE := ET_9STATE_MONITORING.STOPPING;
ELSIF (ENABLE_ON AND STATUS_ON) THEN
	STATE := ET_9STATE_MONITORING.RUNNING;
ELSIF (ENABLE_ON AND STATUS_OFF AND ENABLE_TIMER_ON AND START_DELAY_OFF AND FIRE_OFF) THEN
	STATE := ET_9STATE_MONITORING.STARTING;
ELSIF (ENABLE_OFF AND STATUS_OFF) THEN
	STATE := ET_9STATE_MONITORING.STOPPED;
ELSE
	STATE := ET_9STATE_MONITORING.UNKNOWN;
END_IF;

END_FUNCTION_BLOCK

// DCCM_PLC_1/Application/DEPROX_COUNT
PROGRAM DEPROX_COUNT
VAR
	My_Read_Var: READ_VAR;
	Recieve_Buffer: ARRAY[0..3] OF INT;
	My_Addr_Table: ADDRESS;
	My_Addm: ADDM;
	My_Blink: BLINK;
	My_FLOAT: INT;
	lastValue: INT;
	watchdog: FB_PCMS_WATCHDOG;
END_VAR

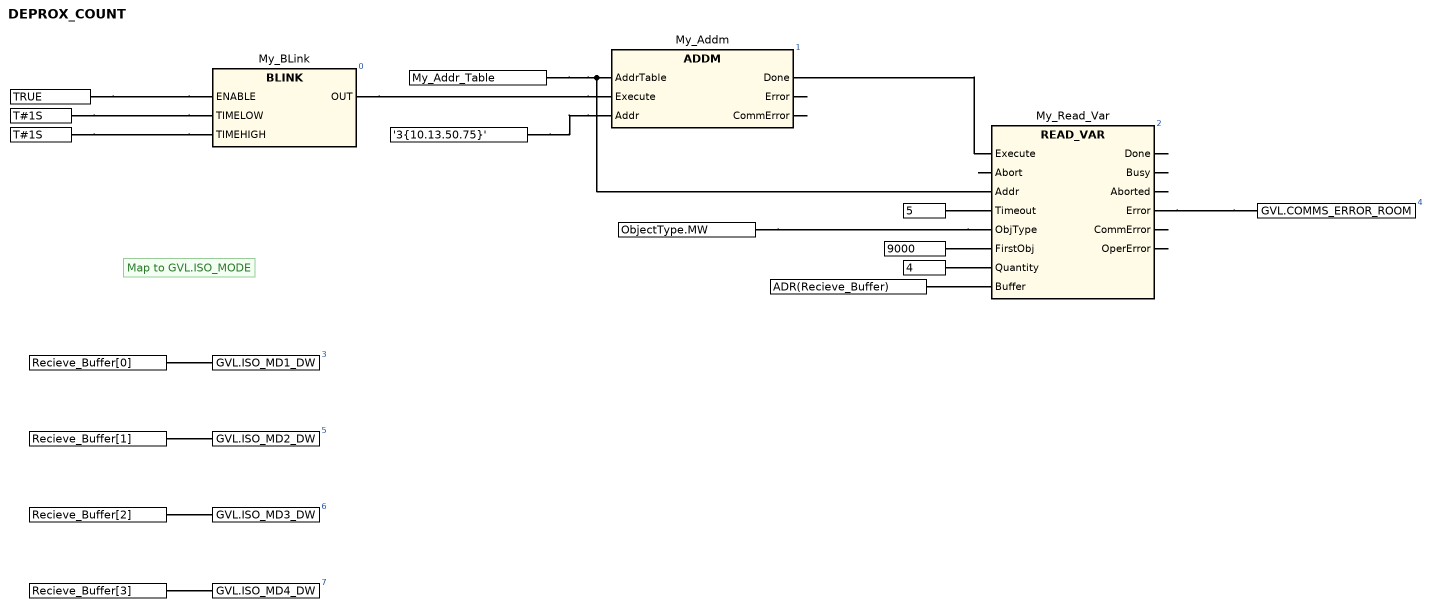
My_BLink(ENABLE := TRUE, TIMELOW := T#1S, TIMEHIGH := T#1S); // BLINK
My_Addm(AddrTable := My_Addr_Table, Execute := My_BLink.OUT, Addr := '3{10.13.50.75}'); // ADDM
My_Read_Var(
    Execute := My_Addm.Done,
    Addr := My_Addr_Table,
    Timeout := 5,
    ObjType := ObjectType.MW,
    FirstObj := 9000,
    Quantity := 4,
    Buffer := ADR(Recieve_Buffer)); // READ_VAR
// Map to GVL.ISO_MODE
GVL.ISO_MD1_DW := Recieve_Buffer[0];
GVL.COMMS_ERROR_ROOM := My_Read_Var.Error;
GVL.ISO_MD2_DW := Recieve_Buffer[1];
GVL.ISO_MD3_DW := Recieve_Buffer[2];
GVL.ISO_MD4_DW := Recieve_Buffer[3];

END_PROGRAM

// DCCM_PLC_1/Application/Library/FB_PCMS_WATCHDOG
FUNCTION_BLOCK FB_PCMS_WATCHDOG
VAR_OUTPUT
	LAST_VALUE: INT;
END_VAR
VAR_INPUT
	VALUE: INT;
END_VAR
VAR_OUTPUT
	TIMEOUT: BOOL;
END_VAR
VAR
	START_DELAY_TON: TON;
END_VAR

START_DELAY_TON(IN := (LAST_VALUE = VALUE), PT := T#120S);
TIMEOUT := START_DELAY_TON.Q;

LAST_VALUE := VALUE;

END_FUNCTION_BLOCK

// DCCM_PLC_1/Application/FAN_2STAGES
PROGRAM FAN_2STAGES
VAR
	FAN_SPEED_PID: PID;
	FAN_SPEED: REAL;
	RTC: SysTimeRtc.RTS_SYSTIMEDATE;
	SysTimeRtcGetResult: UDINT;
	R_TRIG_1: R_TRIG;
	DURY_TRIGGER: FB_DUTYTRIGGER;
	AUTO_STANDBY_FAN_NO: INT;
	FA_2STAGES: FB_2STAGES_DUTY;
	FAN1_EN_LOCAL: BOOL;
	FAN2_SPEED_LOCAL: REAL;
	FAN1_SPEED_LOCAL: REAL;
	FAN2_EN_LOCAL: BOOL;
	VelCheck: TON;
	SR_1: SR;
	TON_FAN1: TON;
	TON_FAN2: TON;
	SR_FAN1: SR;
	SR_FAN2: SR;
	FB_Fan1: FB_FanProvingSwitchOverEnable;
	FB_Fan2: FB_FanProvingSwitchOverEnable;
	DEPROX_COUNT: INT := 0;
	LINEAR_0: LINEAR;
	LINEAR_1: LINEAR;
	SWITCH_CHECK_0: SWITCH_CHECK;
	SWITCH_CHECK_1: SWITCH_CHECK;
	a: BOOL;
	TON_0: TON;
	TON_1: TON;
END_VAR
VAR // added by the converter: edge detectors and wires of the graphical bodies
    _rt1 : R_TRIG;
    _w1, _w2 : BOOL;
END_VAR

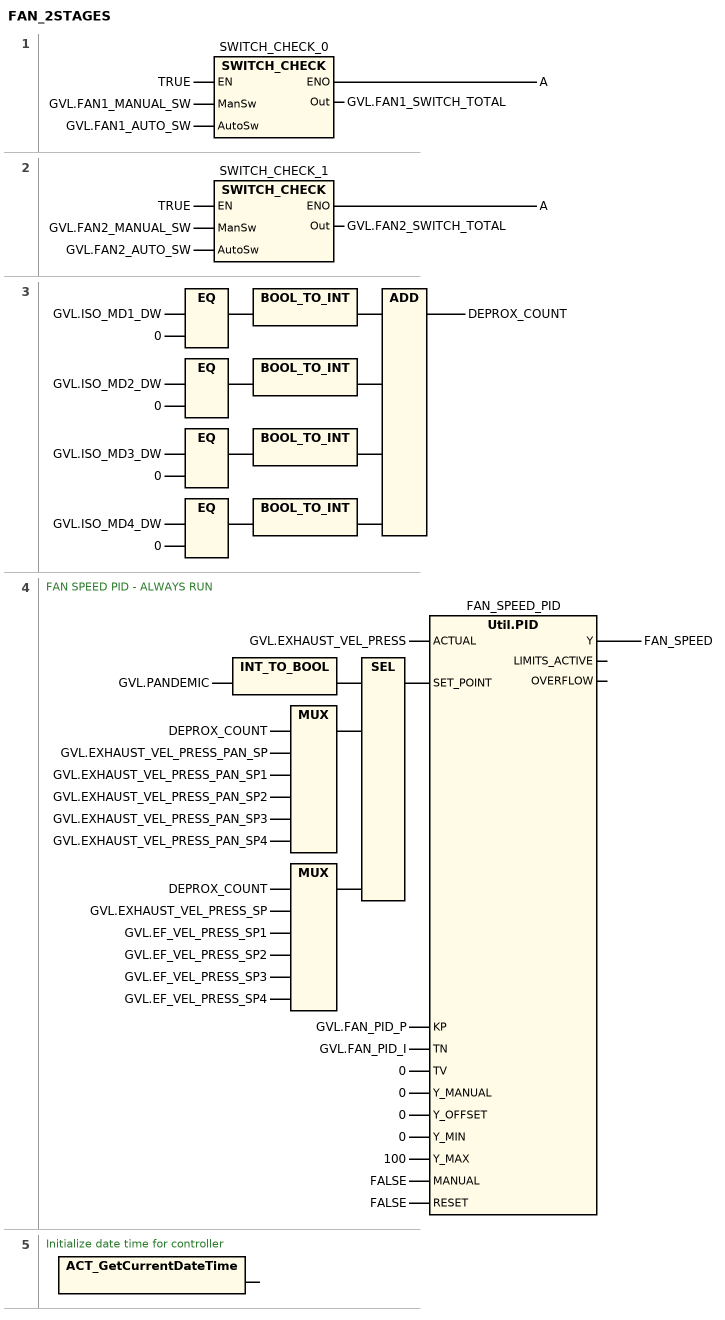
// NETWORK 1
SWITCH_CHECK_0(ManSw := GVL.FAN1_MANUAL_SW, AutoSw := GVL.FAN1_AUTO_SW, Out => GVL.FAN1_SWITCH_TOTAL); // SWITCH_CHECK
A := TRUE;

// NETWORK 2
SWITCH_CHECK_1(ManSw := GVL.FAN2_MANUAL_SW, AutoSw := GVL.FAN2_AUTO_SW, Out => GVL.FAN2_SWITCH_TOTAL); // SWITCH_CHECK
A := TRUE;

// NETWORK 3
DEPROX_COUNT := BOOL_TO_INT(GVL.ISO_MD1_DW = 0) + BOOL_TO_INT(GVL.ISO_MD2_DW = 0) + BOOL_TO_INT(GVL.ISO_MD3_DW = 0) + BOOL_TO_INT(GVL.ISO_MD4_DW = 0);

// NETWORK 4
// FAN SPEED PID - ALWAYS RUN
FAN_SPEED_PID(
    ACTUAL := GVL.EXHAUST_VEL_PRESS,
    SET_POINT := SEL(INT_TO_BOOL(GVL.PANDEMIC), MUX(DEPROX_COUNT, GVL.EXHAUST_VEL_PRESS_PAN_SP, GVL.EXHAUST_VEL_PRESS_PAN_SP1, GVL.EXHAUST_VEL_PRESS_PAN_SP2, GVL.EXHAUST_VEL_PRESS_PAN_SP3, GVL.EXHAUST_VEL_PRESS_PAN_SP4), MUX(DEPROX_COUNT, GVL.EXHAUST_VEL_PRESS_SP, GVL.EF_VEL_PRESS_SP1, GVL.EF_VEL_PRESS_SP2, GVL.EF_VEL_PRESS_SP3, GVL.EF_VEL_PRESS_SP4)),
    KP := GVL.FAN_PID_P,
    TN := GVL.FAN_PID_I,
    TV := 0,
    Y_MANUAL := 0,
    Y_OFFSET := 0,
    Y_MIN := 0,
    Y_MAX := 100,
    MANUAL := FALSE,
    RESET := FALSE); // Util.PID
FAN_SPEED := FAN_SPEED_PID.Y;

// NETWORK 5
// Initialize date time for controller
ACT_GetCurrentDateTime();

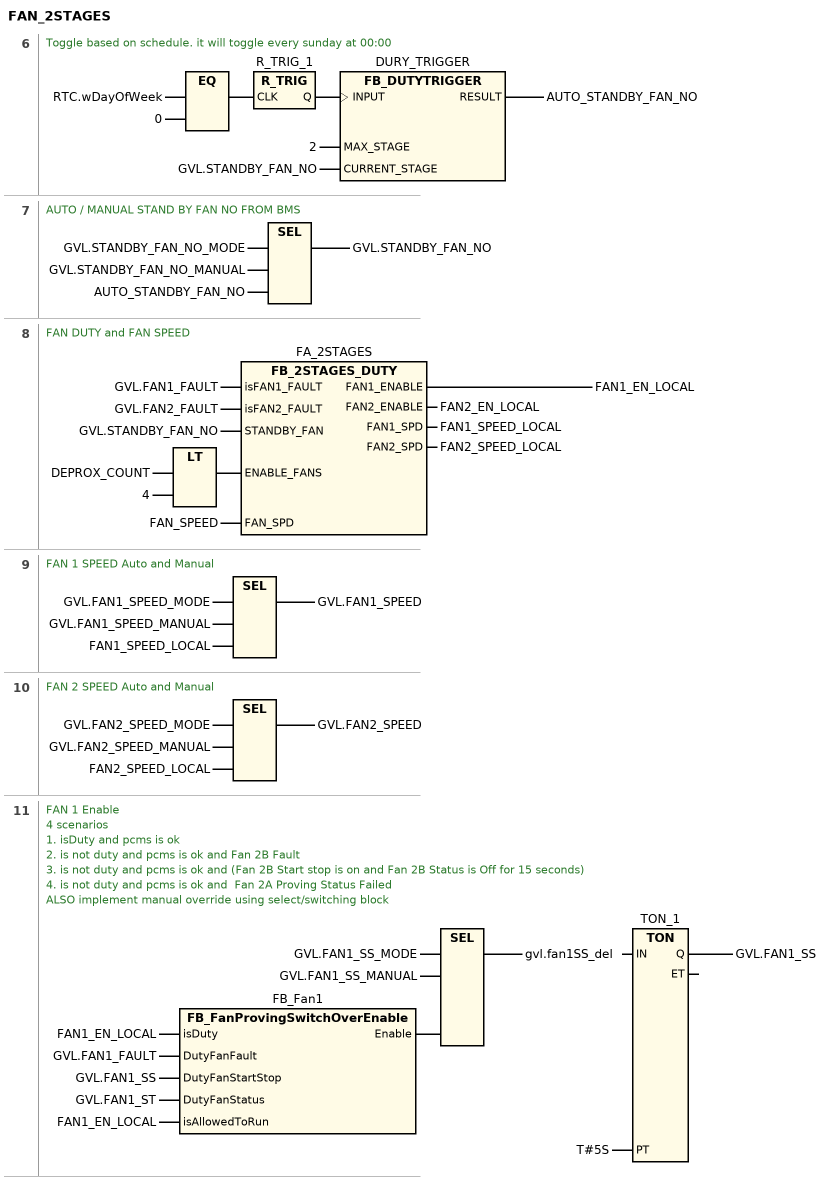
// NETWORK 6
// Toggle based on schedule. it will toggle every sunday at 00:00
R_TRIG_1(CLK := RTC.wDayOfWeek = 0); // R_TRIG
_rt1(CLK := R_TRIG_1.Q);
DURY_TRIGGER(INPUT := _rt1.Q, MAX_STAGE := 2, CURRENT_STAGE := GVL.STANDBY_FAN_NO); // FB_DUTYTRIGGER
AUTO_STANDBY_FAN_NO := DURY_TRIGGER.RESULT;

// NETWORK 7
// AUTO / MANUAL STAND BY FAN NO FROM BMS
GVL.STANDBY_FAN_NO := SEL(GVL.STANDBY_FAN_NO_MODE, GVL.STANDBY_FAN_NO_MANUAL, AUTO_STANDBY_FAN_NO);

// NETWORK 8
// FAN DUTY and FAN SPEED
FA_2STAGES(
    isFAN1_FAULT := GVL.FAN1_FAULT,
    isFAN2_FAULT := GVL.FAN2_FAULT,
    STANDBY_FAN := GVL.STANDBY_FAN_NO,
    ENABLE_FANS := DEPROX_COUNT < 4,
    FAN_SPD := FAN_SPEED,
    FAN2_ENABLE => FAN2_EN_LOCAL,
    FAN1_SPD => FAN1_SPEED_LOCAL,
    FAN2_SPD => FAN2_SPEED_LOCAL); // FB_2STAGES_DUTY
FAN1_EN_LOCAL := FA_2STAGES.FAN1_ENABLE;

// NETWORK 9
// FAN 1 SPEED Auto and Manual
GVL.FAN1_SPEED := SEL(GVL.FAN1_SPEED_MODE, GVL.FAN1_SPEED_MANUAL, FAN1_SPEED_LOCAL);

// NETWORK 10
// FAN 2 SPEED Auto and Manual
GVL.FAN2_SPEED := SEL(GVL.FAN2_SPEED_MODE, GVL.FAN2_SPEED_MANUAL, FAN2_SPEED_LOCAL);

// NETWORK 11
// FAN 1 Enable
// 4 scenarios
// 1. isDuty and pcms is ok
// 2. is not duty and pcms is ok and Fan 2B Fault
// 3. is not duty and pcms is ok and (Fan 2B Start stop is on and Fan 2B Status is Off for 15 seconds)
// 4. is not duty and pcms is ok and  Fan 2A Proving Status Failed
//
// ALSO implement manual override using select/switching block
FB_Fan1(
    isDuty := FAN1_EN_LOCAL,
    DutyFanFault := GVL.FAN1_FAULT,
    DutyFanStartStop := GVL.FAN1_SS,
    DutyFanStatus := GVL.FAN1_ST,
    isAllowedToRun := FAN1_EN_LOCAL); // FB_FanProvingSwitchOverEnable
_w1 := SEL(GVL.FAN1_SS_MODE, GVL.FAN1_SS_MANUAL, FB_Fan1.Enable);
gvl.fan1SS_del := _w1;
TON_1(IN := _w1, PT := T#5S); // TON
GVL.FAN1_SS := TON_1.Q;

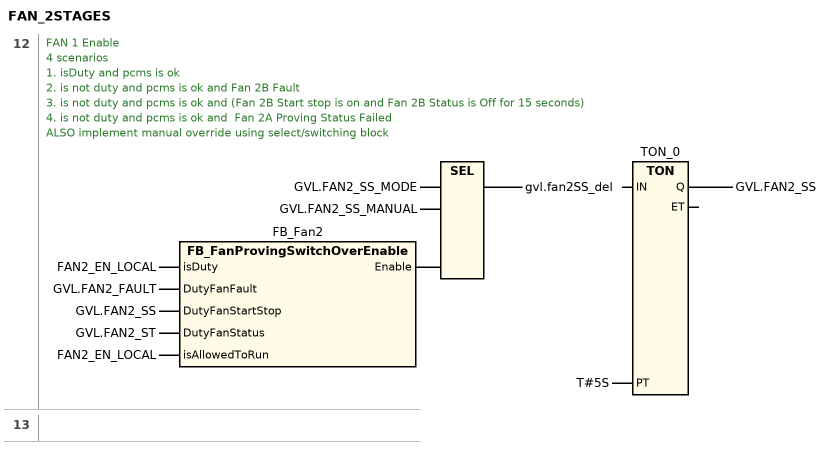
// NETWORK 12
// FAN 1 Enable
// 4 scenarios
// 1. isDuty and pcms is ok
// 2. is not duty and pcms is ok and Fan 2B Fault
// 3. is not duty and pcms is ok and (Fan 2B Start stop is on and Fan 2B Status is Off for 15 seconds)
// 4. is not duty and pcms is ok and  Fan 2A Proving Status Failed
//
// ALSO implement manual override using select/switching block
FB_Fan2(
    isDuty := FAN2_EN_LOCAL,
    DutyFanFault := GVL.FAN2_FAULT,
    DutyFanStartStop := GVL.FAN2_SS,
    DutyFanStatus := GVL.FAN2_ST,
    isAllowedToRun := FAN2_EN_LOCAL); // FB_FanProvingSwitchOverEnable
_w2 := SEL(GVL.FAN2_SS_MODE, GVL.FAN2_SS_MANUAL, FB_Fan2.Enable);
gvl.fan2SS_del := _w2;
TON_0(IN := _w2, PT := T#5S); // TON
GVL.FAN2_SS := TON_0.Q;

// NETWORK 13

ACTION ACT_GetCurrentDateTime:
//you will need to install "SysTimeRtc" library on Application Node -> tools tree

SysTimeRtc.SysTimeRtcConvertUtcToDate( dwTimestampUtc:= SysTimeRtc.SysTimeRtcGet( pResult:= SysTimeRtcGetResult ), pDate:= RTC );
END_ACTION

END_PROGRAM

// DCCM_PLC_1/Application/FBs/SWITCH_CHECK
FUNCTION_BLOCK SWITCH_CHECK
VAR_INPUT
	ManSw: BOOL;
	AutoSw: BOOL;
END_VAR
VAR_OUTPUT
		Out: INT;
END_VAR


Out:=0;

IF ManSw THEN
	Out := 1;
	ELSIF AutoSw THEN
		Out := 2;
END_IF

END_FUNCTION_BLOCK

// DCCM_PLC_1/Application/FBs/FB_DUTYTRIGGER
FUNCTION_BLOCK FB_DUTYTRIGGER
VAR_INPUT
	INPUT: BOOL;
	MAX_STAGE: INT := 2;
	CURRENT_STAGE: INT;
END_VAR
VAR_OUTPUT
	RESULT: INT;
END_VAR

IF(INPUT) THEN
	RESULT := CURRENT_STAGE + 1;
END_IF;

IF(RESULT > MAX_STAGE) OR (RESULT <= 0) THEN
	RESULT:= 1;
END_IF;

END_FUNCTION_BLOCK

// DCCM_PLC_1/Application/FBs/FB_2STAGES_DUTY
FUNCTION_BLOCK FB_2STAGES_DUTY
VAR_INPUT
	isFAN1_FAULT: BOOL;
	isFAN2_FAULT: BOOL;
	STANDBY_FAN: INT := 2;
	ENABLE_FANS: BOOL;
	FAN_SPD: REAL;
END_VAR
VAR_OUTPUT
	FAN1_ENABLE: BOOL;
	FAN2_ENABLE: BOOL;
	FAN1_SPD: REAL;
	FAN2_SPD: REAL;
END_VAR

IF ENABLE_FANS THEN
	IF (STANDBY_FAN = 1) THEN
		IF(isFAN2_FAULT) THEN
			FAN1_ENABLE := TRUE;
			FAN1_SPD := FAN_SPD;
		ELSE
			FAN1_ENABLE := FALSE;
			FAN1_SPD := 0.0;
		END_IF;
		FAN2_ENABLE := TRUE;
		FAN2_SPD := FAN_SPD;
	ELSIF (STANDBY_FAN = 2) THEN
		IF(isFAN1_FAULT) THEN
			FAN2_ENABLE := TRUE;
			FAN2_SPD := FAN_SPD;
		ELSE
			FAN2_ENABLE := FALSE;
			FAN2_SPD := 0.0;
		END_IF;
		FAN1_ENABLE := TRUE;
		FAN1_SPD := FAN_SPD;
	END_IF;
ELSE
	FAN1_ENABLE := FALSE;
	FAN1_SPD := 0.0;
	FAN2_ENABLE := FALSE;
	FAN2_SPD := 0.0;
END_IF;

END_FUNCTION_BLOCK

// DCCM_PLC_1/Application/FBs/FB_FanProvingSwitchOverEnable
FUNCTION_BLOCK FB_FanProvingSwitchOverEnable
VAR_INPUT
	isDuty: BOOL;
	DutyFanFault: BOOL;
	DutyFanStartStop: BOOL;
	DutyFanStatus: BOOL;
	// is Allowed to run
	isAllowedToRun: BOOL;
END_VAR
VAR_OUTPUT
	Enable: BOOL;
END_VAR
VAR
	DelayDutyAnomalyDetected: TON;
END_VAR

//FAN 2A Enable
//4 scenarios
//1. isDuty and pcms is ok
//2. is not duty and pcms is ok and duty fan Fault
//3. is not duty and pcms is ok and (duty fan Start stop is on and duty fan Status is Off for 15 seconds)
//4. is NOT duty AND pcms is ok AND  Fan 2A 2B Proving Status Failed

Enable := FALSE;

DelayDutyAnomalyDetected(IN := (DutyFanStartStop AND NOT DutyFanStatus), PT := T#15S);

IF (isDuty AND isAllowedToRun ) THEN //scenario 1
	ENABLE := TRUE;
ELSIF (NOT isDuty AND isAllowedToRun AND DutyFanFault) THEN //scenario 2
	ENABLE := TRUE;
ELSIF (NOT isDuty AND isAllowedToRun AND DelayDutyAnomalyDetected.Q) THEN //scenario 3
	ENABLE := TRUE;
ELSIF (NOT isDuty AND isAllowedToRun) THEN //scenario 4
	ENABLE := TRUE;
END_IF

END_FUNCTION_BLOCK

// DCCM_PLC_1/Application/FBs/DUTY
FUNCTION_BLOCK DUTY
VAR_INPUT
	DUTY_MAN: BOOL;
	DUTY_MD: BOOL;
	TOGGLE: BOOL;
END_VAR
VAR_OUTPUT
	DUTY: BOOL;
END_VAR

IF (TOGGLE AND DUTY = TRUE AND DUTY_MD = FALSE) THEN
	DUTY := FALSE;
ELSIF (TOGGLE AND DUTY = FALSE AND DUTY_MD = FALSE) THEN
	DUTY := TRUE;
ELSE
	DUTY := DUTY_MAN;
END_IF

END_FUNCTION_BLOCK

// DCCM_PLC_1/Application/FBs/LINEAR
FUNCTION_BLOCK LINEAR
VAR_INPUT
	INPUT: REAL;
	X1: REAL;
	Y1: REAL;
	X2: REAL;
	Y2: REAL;
END_VAR
VAR
	M: REAL;
END_VAR
VAR_OUTPUT
	OUTPUT: REAL;
END_VAR

// Y1-Y2 = M(X1-X2)
//M = (Y2-Y1)/(X2-X1)

M := (Y2 - Y1) / (X2 - X1);
OUTPUT := (M * (INPUT - X1)) + Y1;

END_FUNCTION_BLOCK

// DCCM_PLC_1/Application/PandemicCheck
PROGRAM PandemicCheck
VAR
	My_Read_Var: READ_VAR;
	Recieve_Buffer: ARRAY[0..3] OF INT;
	My_Addr_Table: ADDRESS;
	My_Addm: ADDM;
	My_Blink: BLINK;
	My_FLOAT: INT;
	lastValue: INT;
	watchdog: FB_PCMS_WATCHDOG;
END_VAR

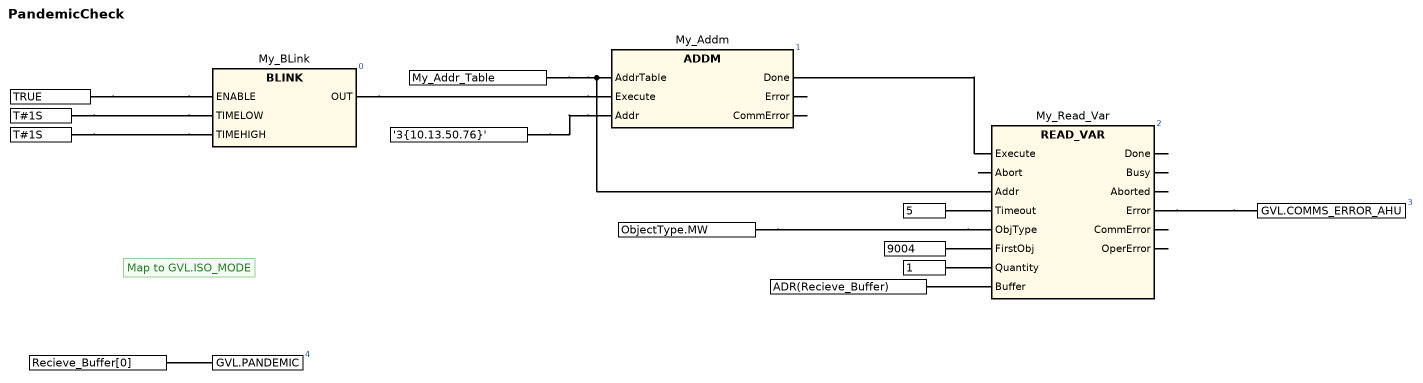
My_BLink(ENABLE := TRUE, TIMELOW := T#1S, TIMEHIGH := T#1S); // BLINK
My_Addm(AddrTable := My_Addr_Table, Execute := My_BLink.OUT, Addr := '3{10.13.50.76}'); // ADDM
My_Read_Var(
    Execute := My_Addm.Done,
    Addr := My_Addr_Table,
    Timeout := 5,
    ObjType := ObjectType.MW,
    FirstObj := 9004,
    Quantity := 1,
    Buffer := ADR(Recieve_Buffer)); // READ_VAR
GVL.COMMS_ERROR_AHU := My_Read_Var.Error;
// Map to GVL.ISO_MODE
GVL.PANDEMIC := Recieve_Buffer[0];

END_PROGRAM

// DCCM_PLC_1/Application/DAMPER_CONTROL
PROGRAM DAMPER_CONTROL
VAR
	A2M_FAN1_DMPR: F_TRIG;
	A2M_FAN2_DMPR: F_TRIG;
	NOT_RUNNING_DELAY: TON;
END_VAR

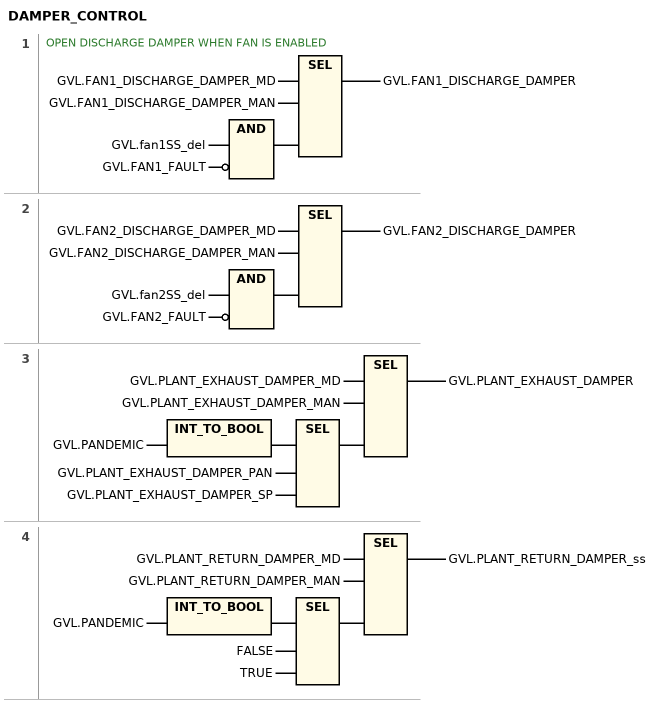
// NETWORK 1
// OPEN DISCHARGE DAMPER WHEN FAN IS ENABLED
GVL.FAN1_DISCHARGE_DAMPER := SEL(GVL.FAN1_DISCHARGE_DAMPER_MD, GVL.FAN1_DISCHARGE_DAMPER_MAN, GVL.fan1SS_del AND NOT GVL.FAN1_FAULT);

// NETWORK 2
GVL.FAN2_DISCHARGE_DAMPER := SEL(GVL.FAN2_DISCHARGE_DAMPER_MD, GVL.FAN2_DISCHARGE_DAMPER_MAN, GVL.fan2SS_del AND NOT GVL.FAN2_FAULT);

// NETWORK 3
GVL.PLANT_EXHAUST_DAMPER := SEL(GVL.PLANT_EXHAUST_DAMPER_MD, GVL.PLANT_EXHAUST_DAMPER_MAN, SEL(INT_TO_BOOL(GVL.PANDEMIC), GVL.PLANT_EXHAUST_DAMPER_PAN, GVL.PLANT_EXHAUST_DAMPER_SP));

// NETWORK 4
GVL.PLANT_RETURN_DAMPER_ss := SEL(GVL.PLANT_RETURN_DAMPER_MD, GVL.PLANT_RETURN_DAMPER_MAN, SEL(INT_TO_BOOL(GVL.PANDEMIC), FALSE, TRUE));

END_PROGRAM

// DCCM_PLC_1/Application/SR_Main
PROGRAM SR_Main
VAR
END_VAR

// NETWORK 1

END_PROGRAM

// DCCM_PLC_1/Application/OUTPUT_MAPPING
PROGRAM OUTPUT_MAPPING
VAR
		voltage_converter: FB_0_10V_TO_2_10V_OUTPUT;
END_VAR

//MAPPING MEMORY WORDS TO HARDWARE OUTPUTS

qFAN1_SPD := TRUNC_INT(GVL.FAN1_SPEED) * 100;									//MODULE 1 TM3AQ4 OUTPUT 0
qFAN2_SPD := TRUNC_INT(GVL.FAN2_SPEED) * 100;									//MODULE 1 TM3AQ4 OUTPUT 1

qFAN1_SS := GVL.FAN1_SS;													//MODULE 3 TM3DM24R OUTPUT 0
qFAN2_SS := GVL.FAN2_SS;													//MODULE 3 TM3DM24R OUTPUT 1

qFAN1_DISCHARGE_DAMPER := NOT GVL.FAN1_DISCHARGE_DAMPER;						//MODULE 3 TM3DM24R OUTPUT 2
qFAN2_DISCHARGE_DAMPER := NOT GVL.FAN2_DISCHARGE_DAMPER;						//MODULE 3 TM3DM24R OUTPUT 3



qPLANT_EXHAUST_DAMPER := REAL_TO_INT((100-GVL.PLANT_EXHAUST_DAMPER) * 100);

qPLANT_RETURN_DAMPER := GVL.PLANT_RETURN_DAMPER_ss;						//CHECK DIRECTION

END_PROGRAM

// DCCM_PLC_1/Application/FBs/DUTY_CHANGE
FUNCTION_BLOCK DUTY_CHANGE
VAR_INPUT
	INPUT: BOOL;
END_VAR
VAR_OUTPUT
	NEW_DUTY: BOOL;
END_VAR
VAR_INPUT
	CURRENT_DUTY: BOOL;
END_VAR

IF INPUT THEN
	IF CURRENT_DUTY = 1 THEN
		NEW_DUTY := 0;
	ELSIF CURRENT_DUTY = 0 THEN
		NEW_DUTY := 1;
	END_IF
END_IF

END_FUNCTION_BLOCK

// DCCM_PLC_1/Application/FBs/FB_DUTY_DUTY_STANDBY_PUMP_SPD
FUNCTION_BLOCK FB_DUTY_DUTY_STANDBY_PUMP_SPD
VAR_INPUT
	SPD_DEM: REAL;
	P1_FLT: BOOL;
	P2_FLT: BOOL;
	P3_FLT: BOOL;
	DUTY: INT;
END_VAR
VAR_OUTPUT
	PUMP1_SPD: REAL;
	PUMP2_SPD: REAL;
	PUMP3_SPD: REAL;
END_VAR

IF (P1_FLT = TRUE AND P2_FLT = TRUE AND P3_FLT = TRUE) THEN				// IF ALL PUMPS IN FAULT, REDUCE SPEED TO 0 FOR ALL PUMPS
	PUMP1_SPD := 0;
	PUMP2_SPD := 0;
	PUMP3_SPD := 0;
ELSIF (DUTY = 0 AND P1_FLT = FALSE AND P2_FLT = FALSE) THEN				//IF PUMP 1 DUTY
	PUMP1_SPD := LIMIT(0, SPD_DEM, 100);
	PUMP2_SPD := LIMIT(0, SPD_DEM - 100, 100);
	PUMP3_SPD := 0;
ELSIF (DUTY = 1 AND P2_FLT = FALSE AND P3_FLT = FALSE)THEN				//IF PUMP 2 DUTY
	PUMP2_SPD := LIMIT(0, SPD_DEM, 100);
	PUMP3_SPD := LIMIT(0, SPD_DEM - 100, 100);
	PUMP1_SPD := 0;
ELSIF(DUTY = 2 AND P3_FLT = FALSE AND P1_FLT = FALSE) THEN				//IF PUMP 3 DUTY
	PUMP3_SPD := LIMIT(0, SPD_DEM, 100);
	PUMP1_SPD := LIMIT(0, SPD_DEM - 100, 100);
	PUMP2_SPD := 0;	
ELSIF (DUTY = 0 AND P1_FLT = TRUE AND P2_FLT = FALSE) THEN				//IF PUMP 1 DUTY AND PUMP 1 IS IN FAULT
	PUMP3_SPD := LIMIT(0, SPD_DEM, 100);
	PUMP2_SPD := LIMIT(0, SPD_DEM - 100, 100);
	PUMP1_SPD := 0;
ELSIF (DUTY = 0 AND P1_FLT = FALSE AND P2_FLT = TRUE) THEN				// IF PUMP 1 DUTY AND PUMP 2 IS IN FAULT
	PUMP1_SPD := LIMIT(0, SPD_DEM, 100);
	PUMP3_SPD := LIMIT(0, SPD_DEM - 100, 100);
	PUMP2_SPD := 0;
ELSIF (DUTY = 0 AND P1_FLT = TRUE AND P2_FLT = TRUE) THEN				//IF PUMP 1 DUTY AND PUMP 1 & 2 ARE IN FAULT
	PUMP3_SPD := LIMIT(0, SPD_DEM, 100);
	PUMP1_SPD := 0;
	PUMP2_SPD := 0;
ELSIF (DUTY = 1 AND P2_FLT = TRUE AND P3_FLT = FALSE) THEN				//IF PUMP 2 DUTY AND PUMP 2 IS IN FAULT
	PUMP1_SPD := LIMIT(0, SPD_DEM, 100);
	PUMP3_SPD := LIMIT(0, SPD_DEM - 100, 100);
	PUMP2_SPD := 0;
ELSIF (DUTY = 1 AND P2_FLT = FALSE AND P3_FLT := TRUE) THEN				//IF PUMP 2 DUTY AND PUMP 3 IS IN FAULT
	PUMP2_SPD := LIMIT(0, SPD_DEM, 100);
	PUMP1_SPD := LIMIT(0, SPD_DEM - 100, 100);
	PUMP3_SPD := 0;
ELSIF (DUTY = 1 AND P2_FLT = TRUE AND P3_FLT := TRUE) THEN				//IF PUMP 2 DUTY AND PUMP 2 & 3 ARE IN FAULT
	PUMP1_SPD := LIMIT(0, SPD_DEM, 100);
	PUMP2_SPD := 0;
	PUMP3_SPD := 0;
ELSIF (DUTY = 2 AND P3_FLT = TRUE AND P1_FLT = FALSE) THEN				//IF PUMP 3 DUTY AND PUMP 3 IS IN FAULT 
	PUMP2_SPD := LIMIT(0, SPD_DEM, 100);
	PUMP1_SPD := LIMIT(0, SPD_DEM - 100, 100);
	PUMP3_SPD := 0;
ELSIF (DUTY = 2 AND P3_FLT = FALSE AND P1_FLT = TRUE) THEN				//IF PUMP 3 DUTY AND PUMP 1 IS IN FAULT
	PUMP3_SPD := LIMIT(0, SPD_DEM, 100);
	PUMP2_SPD := LIMIT(0, SPD_DEM - 100, 100);
	PUMP1_SPD := 0;
ELSIF (DUTY = 2 AND P3_FLT = TRUE AND P1_FLT = TRUE) THEN				//IF PUMP 3 DUTY AND PUMP 3 & 1 ARE IN FAULT
	PUMP2_SPD := LIMIT(0, SPD_DEM, 100);
	PUMP3_SPD := 0;
	PUMP1_SPD := 0;
END_IF

END_FUNCTION_BLOCK

// DCCM_PLC_1/Application/FBs/FB_FLOATING_VALVE
FUNCTION_BLOCK FB_FLOATING_VALVE
VAR_INPUT
	VALVE_OUTPUT: REAL;
	VALVE_TIME: TIME;
END_VAR
VAR_OUTPUT
	VALVE_OPEN: BOOL;
	VALVE_CLOSE: BOOL;
END_VAR
VAR
	CURRENT_POS: REAL;
	MOVE_TIME: TIME;
	MOVE_POS: REAL;
	RS_0: RS;
	TON1: TON;
	OPEN_STOP: BOOL;
	TON2: TON;
	CLOSE_STOP: BOOL;
	RS_1: RS;
END_VAR

IF (VALVE_OUTPUT > CURRENT_POS) THEN
	MOVE_POS := VALVE_OUTPUT - CURRENT_POS;
 	MOVE_TIME := TO_TIME(TO_REAL(VALVE_TIME) * (MOVE_POS / 100)); 
	VALVE_OPEN := TRUE;
	TON1(IN := VALVE_OPEN, PT := MOVE_TIME);
	OPEN_STOP := TON1.Q;
	//RS_0(SET := VALVE_OPEN, RESET1 := OPEN_STOP);
	IF (OPEN_STOP = TRUE) THEN
		VALVE_OPEN := FALSE;
		CURRENT_POS := VALVE_OUTPUT;
	END_IF  
ELSIF (VALVE_OUTPUT < CURRENT_POS) THEN
	MOVE_POS := CURRENT_POS - VALVE_OUTPUT;
	MOVE_TIME := TO_TIME(TO_REAL(VALVE_TIME) * (MOVE_POS / 100));
	VALVE_CLOSE := TRUE;
	TON2(IN := VALVE_CLOSE, PT := MOVE_TIME);
	CLOSE_STOP := TON2.Q;
	//RS_1(SET := VALVE_OPEN, RESET1 := CLOSE_STOP);
	IF (CLOSE_STOP = TRUE) THEN
		VALVE_CLOSE := FALSE;
		CURRENT_POS := VALVE_OUTPUT;
	END_IF
ELSE
	VALVE_OPEN := FALSE;
	VALVE_CLOSE := FALSE;
END_IF

END_FUNCTION_BLOCK

// DCCM_PLC_1/Application/FBs/FB_HEATING_OR_COOLING
FUNCTION_BLOCK FB_HEATING_OR_COOLING
VAR_INPUT
	SAT: REAL;
	SATSP: REAL;
	DB: REAL;
END_VAR
VAR_OUTPUT
	ENABLE_HEATING: BOOL;
	ENABLE_COOLING: BOOL;
END_VAR
VAR_INPUT
	RUN: BOOL;
	HV: REAL;
	CV: REAL;
END_VAR

IF (SAT >= (SATSP + DB) AND RUN AND HV = 0) THEN
	ENABLE_COOLING := TRUE AND ENABLE_HEATING := FALSE;
ELSIF (SAT <= (SATSP - DB) AND RUN AND CV = 0) THEN
	ENABLE_COOLING := FALSE AND ENABLE_HEATING := TRUE;
ELSE
	ENABLE_COOLING := FALSE AND ENABLE_HEATING := FALSE;	
END_IF

END_FUNCTION_BLOCK

// DCCM_PLC_1/Application/FBs/FB_OMODE
FUNCTION_BLOCK FB_OMODE
VAR_INPUT
	ENABLE_BY_TP: BOOL;
	ENABLE_BY_PIR: BOOL;
	ENABLE_BY_AHRS: BOOL;
	MODE: BOOL;
	OMODE_MANUAL: ET_OMODE;
	TPTYPE: BOOL;
END_VAR
VAR_OUTPUT
	OMODE: ET_OMODE;
END_VAR




IF (MODE) THEN
	IF (ENABLE_BY_TP) THEN				//AUTO MODE
		OMODE := ET_OMODE.SCH;
	ELSIF (ENABLE_BY_AHRS) THEN
		OMODE := ET_OMODE.AHRS;
	ELSIF (ENABLE_BY_PIR) THEN
		OMODE := ET_OMODE.MOTDETECT;
	ELSIF (TPTYPE) THEN
		OMODE := ET_OMODE.UNOCC;
	ELSE
		OMODE := ET_OMODE.SETBACK;
	END_IF
ELSE
	OMODE := OMODE_MANUAL;				//MANUAL MODE
END_IF

END_FUNCTION_BLOCK

// DCCM_PLC_1/Application/FBs/FB_PMODE
FUNCTION_BLOCK FB_PMODE
VAR_INPUT
	OMODE: ET_OMODE;
	IS_NOT_SMOKE: BOOL := TRUE;
	FIRE: BOOL;
	PCMS_SIGNAL: INT;
	PCMS_PRIMARY: INT;
	PCMS_MODE: BOOL := TRUE;
	IS_DAMPER_LOCK: BOOL;
	IS_DAMPER_RESET: BOOL;
	IS_PURGE_RUN: BOOL;
	IS_DAMPER_STARTED: BOOL;
	PMODE_MODE: BOOL := TRUE;
	PMODE_MANUAL: ET_PMODE;
END_VAR
VAR_OUTPUT
	AHU_ENABLE: BOOL;
	PMODE: ET_PMODE;
END_VAR

(*  
	Version 1.0
	Last modified: 15/8/2022
	Operating theater mode
	PLEASE USE  FOR OPERATING THEATER ONLY
	IT DOES NOT IMPLEMENT UNOCC, OP_START MODE
	
	OFF_NORMAL := 0,
	OFF_PCMS := 1,
	OFF_FIRE := 2,
	OFF_DMPRLCK := 3,
	OFF_RESET := 4,
	STARTUP := 5,
	RUN_PUR := 6,
	RUN_NORMAL := 7
*)


IF (PMODE_MODE) THEN
	IF (FIRE) THEN
		PMODE := ET_PMODE.OFF_Fire;
	ELSIF (IS_DAMPER_LOCK) THEN
		PMODE := ET_PMODE.OFF_DMPRLOCK;
	ELSIF ((ABS(PCMS_SIGNAL) >= ABS(PCMS_PRIMARY)) AND PCMS_MODE) THEN
		PMODE := ET_PMODE.OFF_PCMS;
	ELSIF (IS_DAMPER_RESET) THEN
		PMODE := ET_PMODE.OFF_RESET;
	ELSIF (IS_PURGE_RUN) THEN
		PMODE := ET_PMODE.Purge;
	ELSIF (IS_DAMPER_STARTED) THEN
		PMODE := ET_PMODE.RUN_NORMAL;
	END_IF
ELSE
	PMODE := PMODE_MANUAL;
END_IF;

AHU_ENABLE := (PMODE = ET_PMODE.Startup OR PMODE = ET_PMODE.Purge OR PMODE = ET_PMODE.RUN_NORMAL) AND IS_NOT_SMOKE = FALSE AND OMODE <> ET_OMODE.UNOCC;

END_FUNCTION_BLOCK

// DCCM_PLC_1/Application/LIBRARY/FB_PULSE_GENERATOR
FUNCTION_BLOCK FB_PULSE_GENERATOR
VAR_INPUT
	ENABLE: BOOL;
END_VAR
VAR_OUTPUT
	OUTPUT: BOOL;
END_VAR
VAR
	PULSESTATE: BOOL;
	PULSETIME: INT;
END_VAR


IF (ENABLE) THEN
	IF(PULSETIME > 100) THEN
		PULSESTATE := NOT PULSESTATE;
		PULSETIME := 0;
	END_IF;
	IF (PULSETIME < 0) THEN
		PULSETIME := 0;
	END_IF;
ELSE
	PULSESTATE := FALSE;
	PULSETIME := 0;
END_IF;

PULSETIME := PULSETIME +1;

OUTPUT := PULSESTATE;

END_FUNCTION_BLOCK

// DCCM_PLC_1/Application/FBs/FB_SETPOINT_MODE
FUNCTION_BLOCK FB_SETPOINT_MODE
VAR_INPUT
	OMODE: ET_OMODE;
	PMODE: ET_PMODE;
	DAY_SP: REAL;
	SETBACK_SP: REAL;
	PURGE_SP: REAL;
END_VAR
VAR_OUTPUT
	RESULT: REAL;
END_VAR

(*
//calculate set point based on plant mode and occupancy mode
	/*
	//occupancy mode
	UNOCC := 0,
	OP_START := 1,
	SCH := 2,
	AHRS := 3,
	MOT_DETECT := 4,
	REVERSE1 := 5,
	REVERSE2 := 6,
	SETBACK := 7,
	
	//plant mode
	OFF_NORMAL := 0,
	OFF_PCMS := 1,
	OFF_FIRE := 2,
	OFF_DMPRLCK := 3,
	OFF_DMPRRESET := 4,
	STARTUP := 5,
	RUN_PUR := 6,
	RUN_NORMAL := 7
	*/
*)

IF (PMODE = ET_PMODE.Purge) THEN
	RESULT := PURGE_SP;
ELSIF ((PMODE = ET_PMODE.RUN_NORMAL) OR (PMODE = ET_PMODE.Startup)) THEN
	IF (OMODE = ET_OMODE.SETBACK) THEN
		RESULT := SETBACK_SP;
	ELSIF(OMODE = ET_OMODE.UNOCC) THEN
		RESULT := 0.0;
	ELSE
		RESULT := DAY_SP;
	END_IF
ELSE
	RESULT := DAY_SP;
END_IF

END_FUNCTION_BLOCK

// DCCM_PLC_1/Application/Library/FB_SETPOINT_RAMPING
FUNCTION_BLOCK FB_SETPOINT_RAMPING
VAR_INPUT
	INPUT: REAL;
	RAMPING_DOWN_TIME_SP: REAL := 10;
	RAMPING_UP_TIME_SP: REAL := 10;
END_VAR
VAR_OUTPUT
	OUTPUT: REAL := 0;
END_VAR
VAR
	TIMER: TON;
	INCREMENT: REAL;
	INPUT_MEMORY: REAL;
END_VAR

(* Set point Ramping up and down *)
IF (OUTPUT = 0) THEN
	OUTPUT := INPUT;
END_IF;

//find the incerement value
IF(INPUT <> INPUT_MEMORY) THEN 
	INPUT_MEMORY := INPUT;	
	IF (INPUT_MEMORY > OUTPUT) THEN
		INCREMENT := (INPUT_MEMORY - OUTPUT)/RAMPING_UP_TIME_SP;
	ELSIF (INPUT_MEMORY < OUTPUT) THEN
		INCREMENT := (INPUT_MEMORY - OUTPUT)/RAMPING_DOWN_TIME_SP;
	ELSE
		INCREMENT := 0;
	END_IF;
END_IF;


IF(INCREMENT <> 0) THEN
	TIMER(IN := NOT TIMER.Q, PT := T#1S);

	IF (TIMER.Q) THEN
		OUTPUT := OUTPUT + INCREMENT;
	END_IF;
	
	IF(OUTPUT > INPUT_MEMORY) AND (INCREMENT > 0) THEN
		//make sure that the output is not over than ouput
		INCREMENT := 0;
		OUTPUT := INPUT_MEMORY;
	ELSIF (OUTPUT < INPUT_MEMORY) AND (INCREMENT < 0) THEN
		//make sure that the output is not less than input
		INCREMENT := 0;
		OUTPUT := INPUT_MEMORY;
	END_IF;
END_IF;

END_FUNCTION_BLOCK

// DCCM_PLC_1/Application/FBs/FB_WATCHDOG
FUNCTION_BLOCK FB_WATCHDOG
VAR_OUTPUT
	LAST_VALUE: INT;
END_VAR
VAR_INPUT
	VALUE: INT;
END_VAR
VAR_OUTPUT
	TIMEOUT: BOOL;
END_VAR
VAR
	START_DELAY_TON: TON;
END_VAR

START_DELAY_TON(IN := (LAST_VALUE = VALUE), PT := T#120S);
TIMEOUT := START_DELAY_TON.Q;

LAST_VALUE := VALUE;

END_FUNCTION_BLOCK

// DCCM_PLC_1/Application/FBs/SATSP_CALC
FUNCTION_BLOCK SATSP_CALC
VAR_INPUT
	SATSP_MID: REAL;
	SATSP_MIN: REAL;
	SATSP_MAX: REAL;
	TL: REAL;
END_VAR
VAR_OUTPUT
	SATSP: REAL;
END_VAR
VAR
	M: REAL;
END_VAR

IF TL > 0 THEN
	M := (SATSP_MID - SATSP_MIN) / 100.0;
	SATSP := (M * (TL)) + SATSP_MIN;
ELSIF TL < 0 THEN
	M := (SATSP_MAX - SATSP_MID) / 100.0;
	SATSP := (M * ABS(TL)) + SATSP_MID;
ELSE
	SATSP := SATSP_MID;
END_IF;

END_FUNCTION_BLOCK

// DCCM_PLC_1/Application/FBs/SB_HEATING_COOLING
FUNCTION_BLOCK SB_HEATING_COOLING
VAR_INPUT
	ENABLE_COOLING: BOOL;
	ENABLE_HEATING: BOOL;
	SATSP: REAL;
	COOLING_SP: REAL;
	HEATING_SP: REAL;
END_VAR
VAR_OUTPUT
	OUT: REAL;
END_VAR
VAR_INPUT
	OMODE: ET_OMODE;
END_VAR

IF (ENABLE_COOLING AND OMODE = ET_OMODE.SETBACK) THEN
	OUT := COOLING_SP;
ELSIF (ENABLE_HEATING AND OMODE = ET_OMODE.SETBACK) THEN
	OUT := HEATING_SP;
ELSE
	OUT := SATSP;
END_IF

END_FUNCTION_BLOCK

// DCCM_PLC_1/Application/SYSTEM_DATE_TIME
PROGRAM SYSTEM_DATE_TIME
VAR
	SysTimeRtcGetResult: UDINT;
	SYS_CLOCK: SysTimeRtc.RTS_SYSTIMEDATE;
END_VAR

//The following program initializes the system date time clock for the PLC. The date/time is subject to variance based on the temperature of the PLC, however this should not cause significant variance unless specific timing is required.
//For the sake of this project, the internal system clock is used for the duty change, tank turnover, etc. - Corey 21.07.2021

//Initializing the system date time
SysTimeRtc.SysTimeRtcConvertUtcToDate( dwTimestampUtc:= SysTimeRtc.SysTimeRtcGet( pResult:= SysTimeRtcGetResult ), pDate:= SYS_CLOCK );

//Updating the global variables for the date, hour and minute using the updated system time.
GVL.SYS_DAY := SYS_CLOCK.wDayOfWeek;
GVL.SYS_HOUR := SYS_CLOCK.wHour;
GVL.SYS_MINUTE := SYS_CLOCK.wMinute;

END_PROGRAM

// DCCM_PLC_1/Application/FBs/TERMINAL_LOAD
FUNCTION_BLOCK TERMINAL_LOAD
VAR_INPUT
	RMT: REAL;
	RMTSP: REAL;
END_VAR
VAR_OUTPUT
	TL: REAL;
END_VAR
VAR_INPUT
	COOL_TL: REAL;
	HEAT_TL: REAL;
END_VAR

IF (RMTSP > RMT) THEN
	TL := (-1.0 * HEAT_TL);
ELSE
	TL := COOL_TL;	
END_IF;

END_FUNCTION_BLOCK

// DCCM_PLC_1/Application/FBs/FB_2STAGES_DUTY_1
FUNCTION_BLOCK FB_2STAGES_DUTY_1

VAR_INPUT
	isFAN1_FAULT : BOOL;
	isFAN2_FAULT : BOOL;
	STANDBY_FAN : INT := 1;
	ENABLE_FANS : BOOL;
	FAN_SPD : REAL;
END_VAR

VAR_OUTPUT
	FAN1_ENABLE : BOOL;
	FAN2_ENABLE : BOOL;
	FAN1_SPD : REAL;
	FAN2_SPD : REAL;
END_VAR

IF ENABLE_FANS THEN
	IF (STANDBY_FAN = 1) THEN
		IF(isFAN2_FAULT) THEN
			FAN1_ENABLE := TRUE;
			FAN1_SPD := FAN_SPD;
		ELSE
			FAN1_ENABLE := FALSE;
			FAN1_SPD := 0.0;
		END_IF;
		FAN2_ENABLE := TRUE;
		FAN2_SPD := FAN_SPD;
	ELSIF (STANDBY_FAN = 2) THEN
		IF(isFAN1_FAULT) THEN
			FAN2_ENABLE := TRUE;
			FAN2_SPD := FAN_SPD;
		ELSE
			FAN2_ENABLE := FALSE;
			FAN2_SPD := 0.0;
		END_IF;
		FAN1_ENABLE := TRUE;
		FAN1_SPD := FAN_SPD;
	END_IF;
ELSE
	FAN1_ENABLE := FALSE;
	FAN1_SPD := 0.0;
	FAN2_ENABLE := FALSE;
	FAN2_SPD := 0.0;
END_IF;

END_FUNCTION_BLOCK
